# EPICS autosave request: tests/testfiles/cfg/SF_RF_PV.req
$(SYS)-RMSM:SM-SET
$(SYS)-RSYS:REQUIRED-OP
$(SYS)-RILK:MODE-CMD
$(SYS)-RSYS:SET-STATION-STATE
$(SYS)-RSYS:SET-BEAM-PHASE
$(SYS)-RSYS:SET-VSUM-PHASE
$(SYS)-RSYS:SET-KLY-POWER
$(SYS)-RSYS:SET-ACC-VOLT
$(SYS)-RSYS:GET-ACC-VOLT
$(SYS)-RSYS:SET-VSUM-PHASE-OFFSET-BASE
$(SYS)-RSYS:SET-VSUM-AMPLT-SCALE
$(SYS)-RSYS:SET-VOLT-POWER-SCALE
